{attribute addProperty BoxType "EL6688-0000-0017"}
{attribute addProperty Id "Sync_ModeAT %I*BYTE812Control_value_update_toggleAT %I*BOOL8114Time_stamp_update_toggleAT %I*BOOL8115External_device_not_connectedAT %I*BOOL8116Internal_time_stampAT %I*ULINT64817External_time_stampAT %I*ULINT64818Control_Value_for_DC_Master_ClockAT %I*DINT32419"}
{attribute addProperty CRC "2857877896"}
{attribute addProperty SizeInBites "192"}
{attribute addProperty SizeInBytes "24"}
TYPE External_Sync_AA57C188 :
STRUCT
	{attribute addProperty Name "Sync_Mode"}
	Sync_Mode AT %I* : BYTE;
	{attribute addProperty Name "Control_value_update_toggle"}
	Control_value_update_toggle AT %I* : BOOL;
	{attribute addProperty Name "Time_stamp_update_toggle"}
	Time_stamp_update_toggle AT %I* : BOOL;
	{attribute addProperty Name "External_device_not_connected"}
	External_device_not_connected AT %I* : BOOL;
	{attribute addProperty Name "Internal_time_stamp"}
	Internal_time_stamp AT %I* : ULINT;
	{attribute addProperty Name "External_time_stamp"}
	External_time_stamp AT %I* : ULINT;
	{attribute addProperty Name "Control_Value_for_DC_Master_Clock"}
	Control_Value_for_DC_Master_Clock AT %I* : DINT;
END_STRUCT
END_TYPE

(* stored: Version 1.2.0.0, ProductVersion 3.1.4024.9
   DUT External_Sync_AA57C188: Id {ee6dd931-8d69-4456-afbb-53040bd02bd4} *)
